FUNCTION SCALE (* Scaling Function Block *)
  (* Standard: 61499-1; Description: was inspired by this Video: EP2 - CODESYS: Create Scaling Function Block https://www.youtube.com/watch?v=Ir6QAxxDarI *)
  (* Version 1.0, 2024-09-19, franz *)
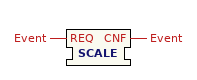
  EVENT_INPUT
    REQ;
  END_EVENT
  EVENT_OUTPUT
    CNF;
  END_EVENT
  BODY IN ST:

  END_BODY
END_FUNCTION
